// TIA Portal V20 export
DATA_BLOCK "Test"   // DB1
{ S7_Optimized_Access := 'TRUE' }
// stored: MemoryReserve 100
   VAR
      testing_bool_output : Bool;
      testing_bool_input : Bool;
      Tag_A : Int := 1;
      Tag_B : Int := 2;
      Tag_C : Int := 3;
      Tag_D : Int := 4;
      Tag_E : Int := 5;
      Testing : Array[0..4] of Int;
   END_VAR
BEGIN
END_DATA_BLOCK
